// TIA Portal project "Project2" (V17)

(* hardware
DEVICE "S7-1200 station_1"  S7-1200 Station
   slot 0: "Rack_0"  S7-1200 Rack  Rack  V1.0
   slot 1: "PLC_1"  CPU 1214C DC/DC/DC  6ES7 214-1AG40-0XB0  V4.5
*)

// ===== PLC "PLC_1"  CPU 1214C DC/DC/DC =====

VAR_GLOBAL   // PLC tag table "Default tag table"
   "start" AT %M0.0 : Bool;
   "stop" AT %M0.1 : Bool;
   "conveyor" AT %M0.2 : Bool;
END_VAR

ORGANIZATION_BLOCK "Main"   // OB1, LAD, ProgramCycle
TITLE = "Main Program Sweep (Cycle)"
{ S7_Optimized_Access := 'TRUE' }
VERSION : 0.1
   VAR_INPUT
      Initial_Call : Bool;   // Initial call of this OB
      Remanence : Bool;   // =True, if remanent data are available
   END_VAR
BEGIN

REGION Network 1
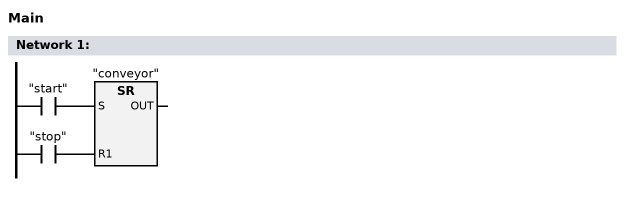
   RUNG wire#powerrail
      Contact( "start" )
      S_SR(operand := "conveyor", r1 := wire#w1)
   END_RUNG
   RUNG wire#powerrail
      Contact( "stop" )
   END_RUNG wire#w1
   // the same network as SCL:
   IF "start" THEN
       "conveyor" := TRUE;   // SR flip-flop
   END_IF;
   IF "stop" THEN "conveyor" := FALSE; END_IF;
END_REGION
END_ORGANIZATION_BLOCK